# EPICS autosave request: iocBoot/generic_motors_ioc/dbSave/XY_P12_.req
%
% BURT Request File
%
% $(P)XY:P12:  X-Y positioner #12
%

file assy.req ASSY=$(P)XY:P12
file mtr1.req MTR1=$(P)XY:mx12
file mtr1.req MTR1=$(P)XY:my12
file drv1.req DRV1=$(P)XY:X12
file drv1.req DRV1=$(P)XY:Y12
